// TIA Portal V18 export
DATA_BLOCK "Pump Manage"   // DB307
{ S7_Optimized_Access := 'TRUE' }
VERSION : 0.1
// stored: AutoNumber true, DBAccessibleFromOPCUA true, IsOnlyStoredInLoadMemory false, IsRetainMemResEnabled false, IsWriteProtectedInAS false, MemoryReserve 100
   VAR RETAIN
      "Pump A-Run Time Hours<50%" : UDInt;
      "Pump A-Run Time Minuts<50%" : UDInt;
      "Pump A-Run Time Seconds<50%" : UDInt;
      "Pump B-Run Time Hours<50%" : UDInt;
      "Pump B-Run Time Minuts<50%" : UDInt;
      "Pump B-Run Time Seconds<50%" : UDInt;
      "Pump A-Run Time Hours>50%" : UDInt;
      "Pump A-Run Time Minuts>50%" : UDInt;
      "Pump A-Run Time Seconds>50%" : UDInt;
      "Pump B-Run Time Hours>50%" : UDInt;
      "Pump B-Run Time Minuts>50%" : UDInt;
      "Pump B-Run Time Seconds>50%" : UDInt;
   END_VAR
   VAR
      "Pump A Min Reset<50" : Bool;
      "Pump A Hrs Reset1<50" : Bool;
      "comm Pump A Hrs Reset<50" : Bool;
      "Pump A Hrs Reset<50" : Bool;
      "Pump A Sec Reset<50" : Bool;
      "Pump A Min Reset>50" : Bool;
      "Pump A Hrs Reset>50" : Bool;
      "Pump A Hrs Reset1>50" : Bool;
      "comm Pump A Hrs Reset>50" : Bool;
      "Pump A Sec Reset>50" : Bool;
      "Pump B Min Reset<50" : Bool;
      "Pump B Hrs Reset<50" : Bool;
      "Pump B Hrs Reset1<50" : Bool;
      "comm Pump B Hrs Reset<50" : Bool;
      "Pump B Sec Reset<50" : Bool;
      "Pump B Min Reset>50" : Bool;
      "Pump B Hrs Reset>50" : Bool;
      "Pump B Hrs Reset1>50" : Bool;
      "comm Pump B Hrs Reset>50" : Bool;
      "Pump B Sec Reset>50" : Bool;
      "Reset A pump Hours and Minutes" : Bool;
      "Reset B pump Hours and Minutes" : Bool;
   END_VAR
   VAR RETAIN
      "Pump A Total Run Hours" : UDInt;
      "Pump B Total Run Hours" : UDInt;
      "Pump A Total Run Minutes" : UDInt;
      "Pump B Total Run Minutes" : UDInt;
   END_VAR
   VAR
      "Pump SEc Reset" : Struct
         "comm Pump A Sec Reset<50" : Bool;
         "comm Pump A Sec Reset>50" : Bool;
         "comm Pump B Sec Reset<50" : Bool;
         "comm Pump B Sec Reset>50" : Bool;
      END_STRUCT;
   END_VAR
BEGIN
END_DATA_BLOCK
